METHOD  M_STATE_RESETTING
VAR_INPUT
END_VAR
Error :=_Error;
Done :=_Executed;
Busy := FALSE;


CASE uiResettingStep OF
	
	0:
		ConveyorMotor.M_MotorStop();
		M_RecoveryAllObjects();
		uiResettingStep:=9999;


	9999:
		M_RecoveryAllObjects();
		_ResetCompleted:=TRUE;
END_CASE
IF _ResetCompleted THEN
	eSTATE:=STATE_DORMANT;
END_IF
END_METHOD

END_FUNCTION_BLOCK

// ---- Library/20_MachineUnits/22_AllocateArea/Old_Version_Service/FB_OutRobot_EmptyBoxMove_old.TcPOU
FUNCTION_BLOCK FB_OutRobot_EmptyBoxMove_old EXTENDS FB_ObjectBase_V2
VAR_INPUT
//    Execute    :BOOL;   // True : This prog will start.
//    Abort      :BOOL;   // True : This prog will be abort.
//    Reset      :BOOL;   // True : This prog will be reset.
//    ObjectName :STRING; // Set this fb name(About it's action)
	INPUT            			   : REFERENCE TO ST_InputTable;
	Cylinder   					   : REFERENCE TO UNI_CylinderList;
	Motor      					   : REFERENCE TO UNI_MotorList;
	AutoMode_OutRobotMoveMove : st_AutoMode_ClampingBoxesJob;	
	Cylinders					   : REFERENCE TO ARRAY[0..1] OF FB_Cylinder;
	Clips						   : REFERENCE TO ARRAY[0..1] OF FB_Cylinder;
END_VAR

VAR_OUTPUT
//    Busy    :BOOL;        // True : This prog is running.
//    Done    :BOOL;        // True : Command has been executed.
//    Aborted :BOOL;        // True : This prog is aborted.
//    Error   :BOOL;        // True : This prog has an error.
//    ErrorID :UINT;       // Output ErrorID
//    Status  :T_MaxString; // Output this prog status by string(255bytes)
END_VAR

VAR
//    eState :E_MethodStatus_Basic;
//	uiExecutingStep : UDINT; // This var is used to been controll STATE_EXECUTING process.
//	uiResettingStep : UDINT;
//	uiAbortingStep : UDINT;
//	_Executed :BOOL; // Executing process completed.
//	_Error : BOOL; // FB has an error.
//	_ResetCompleted : BOOL; // FB resetting completed.
//	_AbortCompleted : BOOL; // FB aborting completed.
	//_Abort		: BOOL;
	strStatus	: STRING;
	uiResumeStep : UINT;
	tonTimeOut   :TON;
	tonTimeDelay   :TON;
	iWorkingIndex : INT;
	_UniqueErrorCode :STRING;	
	
	PickingPos	: ARRAY[0..1] OF ST_PositionTable;
	PlacingPos  : ARRAY[0..1] OF ST_PositionTable;
	PressCylinderOnI5			   : REFERENCE TO FB_Cylinder;
	bSyncPick	: BOOL;
	bSyncPlace	: BOOL;
	SensorOnConveyor		   : BIT;
	ConveyorMotor				   : REFERENCE TO FB_Motor;
	UseA	: BOOL;
	UseB	: BOOL;
END_VAR

A00_BasicUnits();
SUPER^.A10_StateControl();

ACTION A00_BasicUnits:
tonTimeOut(PT:=T#60S);
tonTimeDelay(PT:=T#1s);
END_ACTION

METHOD GetModelState
VAR_OUTPUT
    xDone    :BOOL;
    xBusy    :BOOL;
    xError   :BOOL;
    xAborted :BOOL;
    iErrorID :UDINT;
	UniqueErrorCode : STRING;
END_VAR
xDone    := Done;
xBusy    := Busy;
xError   := Error;
xAborted := Abort;
iErrorID := ErrorID;
UniqueErrorCode := THIS^.UniqueErrorCode;
END_METHOD

METHOD GetName : STRING
GetName := ObjectName;
END_METHOD

METHOD PRIVATE M_CheckCommand : BOOL
VAR_INPUT
END_VAR


M_CheckCommand := true;
END_METHOD

METHOD PRIVATE M_GetWorkingConditions : BOOL
VAR_INPUT
END_VAR
IF AutoMode_OutRobotMoveMove.ClampingInfo.UseClibA THEN
	PickingPos[0] :=FUN_GetPositionTableData('I',5,0);
	PlacingPos[0]:=FUN_GetPositionTableData('R',1,0);
	UseA :=TRUE;
END_IF

IF AutoMode_OutRobotMoveMove.ClampingInfo.UseClibB THEN
	PickingPos[1] :=FUN_GetPositionTableData('I',5,1);
	PlacingPos[1]:=FUN_GetPositionTableData('R',2,1);
	UseB := TRUE;
END_IF

IF PlacingPos[0].X_Pos =PlacingPos[1].X_Pos AND PlacingPos[0].Y_Pos = PlacingPos[1].Y_Pos AND UseA AND UseB  THEN
		bSyncPlace:=TRUE;
	ELSE
		bSyncPlace:=FALSE;	
END_IF
IF PickingPos[0].X_Pos =PickingPos[1].X_Pos AND PickingPos[0].Y_Pos = PickingPos[1].Y_Pos AND UseA AND UseB THEN
		bSyncPick:=TRUE;
	ELSE
		bSyncPick:=FALSE;	
END_IF

PressCylinderOnI5 REF= Cylinder.List.fbDifferentSizeCV_Press2;


ConveyorMotor REF= Motor.List.TransmitDifferentSideCV;
END_METHOD

METHOD PRIVATE M_RecoveryAllObjects : BOOL
VAR_INPUT
END_VAR
VAR 
	i : INT;
END_VAR
FOR i:=0 TO 1 DO
	IF Clips[i].xError THEN
		Clips[i].M_Reset();
		ELSE
		Clips[i].M_Retract();		
	END_IF
	IF Cylinders[i].xError THEN
	Cylinders[i].M_Reset();	
	ELSE
	Cylinders[i].M_Retract();	
	END_IF
END_FOR


IF arAxisCtrl_gb[AxisNo.OutRobot_X].Admin.Axis.Status.Error THEN

	arAxisCtrl_gb[AxisNo.OutRobot_X].Admin.ClearError:= TRUE;
ELSE
	arAxisCtrl_gb[AxisNo.OutRobot_X].Admin.ClearError:= FALSE;
END_IF

IF arAxisCtrl_gb[AxisNo.OutRobot_Y].Admin.Axis.Status.Error THEN

	arAxisCtrl_gb[AxisNo.OutRobot_Y].Admin.ClearError:= TRUE;
ELSE
	arAxisCtrl_gb[AxisNo.OutRobot_Y].Admin.ClearError:= FALSE;
END_IF
END_METHOD

METHOD  M_STATE_ABORTED
VAR_INPUT
END_VAR
ERROR :=TRUE;
Busy    := FALSE;
Aborted := TRUE;
Status := strStatus;

IF NOT Execute THEN
	eSTATE:=STATE_RESETTING;
END_IF

IF Execute AND Reset THEN
//	uiExecutingStep :=uiResumeStep;
	eSTATE:=STATE_EXECUTING;
END_IF
END_METHOD

METHOD  M_STATE_ABORTING
VAR_INPUT
END_VAR
VAR	 
 i : INT;
	bCylinderCheck: BOOL;
END_VAR
Error := TRUE;
CASE uiAbortingStep OF
	0 :
		bCylinderCheck :=TRUE;
		ConveyorMotor.M_MotorStop();
	
		FOR i :=0 TO 1 DO		
	    	Cylinders[i].M_Reset();
			Cylinders[i].M_Retract();
			bCylinderCheck:=bCylinderCheck AND Cylinders[i].InRearPosition;	
		END_FOR
		IF bCylinderCheck THEN		
			uiAbortingStep:=9999;
		END_IF
	9999:	_AbortCompleted:=TRUE;
END_CASE

IF _AbortCompleted THEN	
	eSTATE :=STATE_ABORTED;
END_IF
END_METHOD

METHOD  M_STATE_DONE
VAR_INPUT
END_VAR
Busy 	:= FALSE;
Done	:=TRUE;

IF NOT Execute THEN
	eSTATE:=STATE_RESETTING;
END_IF
END_METHOD

METHOD  M_STATE_DORMANT
VAR_INPUT
END_VAR
Busy            := FALSE;
Done            := FALSE;
Aborted         := FALSE;
Error           := FALSE;
ErrorID         := 0;
Status          := '';
_ResetCompleted := FALSE;
_Error          := FALSE;
_Executed       := FALSE;
_Abort	 :=FALSE;
strStatus :='FB_OutRobot_EmptyBoxMove: No Error';
uiExecutingStep :=uiResettingStep :=uiResumeStep :=0;
tonTimeOut.IN :=TRUE;
_UniqueErrorCode:='0';
iWorkingIndex :=0;
bSyncPlace := FALSE;
UseA := FALSE;
UseB :=FALSE;
IF Execute THEN
	eSTATE:=STATE_EXECUTING;
END_IF
END_METHOD

METHOD  M_STATE_ERROR
VAR_INPUT
END_VAR
ERROR   :=TRUE;
Busy	:=FALSE;
Status := strStatus;
IF __ISVALIDREF(ConveyorMotor) THEN
	ConveyorMotor.M_MotorStop();
END_IF
IF NOT Execute THEN	
eSTATE:=STATE_RESETTING;
END_IF
END_METHOD

METHOD  M_STATE_EXECUTING
VAR_INPUT
END_VAR
VAR_INST
	bMoveConveyorForward : BOOL;
	bMoveConveyorBackrward : BOOL;

END_VAR

VAR
	bCylinderCheck : BOOL := TRUE;
END_VAR
Busy :=TRUE;
SensorOnConveyor := INPUT.bDifferentSizeCV_BoxDetect5_Sensor;
IF bMoveConveyorForward THEN
	IF NOT ConveyorMotor.InBackWard THEN
		ConveyorMotor.M_MoveForward();
	END_IF
END_IF
IF bMoveConveyorBackrward THEN
	IF NOT ConveyorMotor.InForWard THEN
		ConveyorMotor.M_MoveBackward();
	END_IF
END_IF
CASE uiExecutingStep OF
	

0: //Idle
	bMoveConveyorForward:=FALSE;
	bMoveConveyorBackrward:=FALSE;
	tonTimeDelay.IN :=FALSE;
	tonTimeOut.IN := FALSE;
	iWorkingIndex :=0;
	M_GetWorkingConditions();
	
	
	M_RecoveryAllObjects();
	uiExecutingStep := 100;
	
100: //Check command
	
	IF PressCylinderOnI5.xError THEN
		PressCylinderOnI5.M_Reset();
	ELSE
		PressCylinderOnI5.M_Retract();
	END_IF
	
	IF M_CheckCommand() THEN
		uiExecutingStep:=200;
	END_IF
	
200: // Check No boxes turntable

	IF (UseA AND INPUT.bTurnTable_R1Detect_Sensor) OR (UseB AND INPUT.bTurnTable_R2Detect_Sensor) THEN
		_Abort:=TRUE;
		strStatus :='FB_OutRobot_EmptyBoxMove Step 200: Box On Turntable';
	ELSE
		IF UseA THEN
			iWorkingIndex :=0;
		ELSE
			iWorkingIndex :=1;	
		END_IF
		
		uiExecutingStep:=1000;	
	END_IF

	
1000: 
	// Move Conveyor
	// Move OutRobot to First clip picking	
	 //ConveyorMotor.M_MoveForward();
	 bMoveConveyorForward:=TRUE;
	arAxisCtrl_gb[AxisNo.OutRobot_X].PosMode.Position := PickingPos[iWorkingIndex].X_Pos;		
	arAxisCtrl_gb[AxisNo.OutRobot_Y].PosMode.Position := PickingPos[iWorkingIndex].Y_Pos;	
		IF ConveyorMotor.InForWard THEN
			uiExecutingStep:=1100;
		END_IF
		
1100://CheckSensor
	tonTimeDelay.IN:=SensorOnConveyor;
	
			
	IF tonTimeDelay.Q THEN
		tonTimeOut.IN :=FALSE;
		uiExecutingStep:=1200;
		tonTimeDelay.IN := FALSE;
		
	END_IF
	
	tonTimeOut.IN := TRUE;
	IF tonTimeOut.Q THEN
		tonTimeOut.IN :=FALSE;
		_Abort := TRUE;
		strStatus :='FB_OutRobot_EmptyBoxMove Step 1100: No Box on conveyor';
	END_IF

1200: //Press seconde box
	  PressCylinderOnI5.M_Extend();
	  IF PressCylinderOnI5.InFrontPosition THEN
		  tonTimeOut.IN :=FALSE;
		  uiExecutingStep:=1300;
	  END_IF
	  
	  	tonTimeOut.IN := TRUE;
	IF tonTimeOut.Q THEN
		tonTimeOut.IN :=FALSE;
		_Abort := TRUE;
		strStatus :='FB_OutRobot_EmptyBoxMove Step 1200: Block box on conveyor timeout';
	END_IF
	
1300: // Stop conveyor
	ConveyorMotor.M_MotorStop();
	bMoveConveyorForward:=FALSE;
	bMoveConveyorBackrward:=FALSE;
	IF ConveyorMotor.InStopped THEN
		 uiExecutingStep:=1400;
	END_IF

1400: // Check outRobot arrived
	IF		(arAxisStatus_gb[AxisNo.OutRobot_X].Admin._OpModeAck = ModePosAbs AND arAxisStatus_gb[AxisNo.OutRobot_X].Admin.CmdDone) 
	AND (arAxisStatus_gb[AxisNo.OutRobot_Y].Admin._OpModeAck = ModePosAbs AND arAxisStatus_gb[AxisNo.OutRobot_Y].Admin.CmdDone) 
	THEN
		tonTimeOut.IN :=FALSE;
		uiExecutingStep:=1500;
	END_IF	
	
	tonTimeOut.IN := TRUE;
	IF tonTimeOut.Q THEN
		tonTimeOut.IN :=FALSE;
		_Error := TRUE;
		strStatus :='FB_OutRobot_EmptyBoxMove Step 1400: Move robot to picking position timeout';
	END_IF
	
1500: //Clip Down Pick
	 Cylinders[iWorkingIndex].M_Extend();
	  IF Cylinders[iWorkingIndex].InFrontPosition THEN
		  tonTimeOut.IN :=FALSE;
		  uiExecutingStep:=1700;
	  END_IF
	
	 tonTimeOut.IN := TRUE;
	IF tonTimeOut.Q THEN
		tonTimeOut.IN :=FALSE;
		_Abort := TRUE;
		strStatus :='FB_OutRobot_EmptyBoxMove Step 1500: Cylinder pick down timeout';
	END_IF
	
1700: // Clip close Pick
	Clips[iWorkingIndex].M_Extend();
	  IF Clips[iWorkingIndex].InFrontPosition THEN
		  tonTimeOut.IN :=FALSE;
		  uiExecutingStep:=1800;
	  END_IF
	  
	   tonTimeOut.IN := TRUE;
	IF tonTimeOut.Q THEN
		tonTimeOut.IN :=FALSE;
		_Abort := TRUE;
		strStatus :='FB_OutRobot_EmptyBoxMove Step 1700: clip pick close timeout';
	END_IF

1800: // Clip Up Pick
	   Cylinders[iWorkingIndex].M_Retract();
	  IF Cylinders[iWorkingIndex].InRearPosition THEN
		  
		  tonTimeOut.IN :=FALSE;
		  uiExecutingStep:=1850;
	  END_IF
	  
	    tonTimeOut.IN := TRUE;
	IF tonTimeOut.Q THEN
		tonTimeOut.IN :=FALSE;
		_Abort := TRUE;
		strStatus :='FB_OutRobot_EmptyBoxMove Step 1800: cylinder pick up timeout';
	END_IF
1850: //Check box leave
		IF NOT SensorOnConveyor THEN
			PressCylinderOnI5.M_Retract();
			uiExecutingStep:=1900;
		else
			_Error := TRUE;
			strStatus :='FB_OutRobot_EmptyBoxMove Step 1850: Box still on conveyor';
		END_IF
		
1900: // If Next pick
	  IF iWorkingIndex>=1 OR NOT UseB THEN
		  IF UseA THEN
		  	iWorkingIndex :=0;
		  ELSIF UseB THEN
			iWorkingIndex :=1;	
		  END_IF
		  uiExecutingStep:=2000;
		  //Go to placing box
	  ELSIF  iWorkingIndex=0 AND UseB THEN
			iWorkingIndex:=iWorkingIndex+1;
	 		uiExecutingStep:=1000;
	  END_IF
	  
2000: // Move to Placing pos
	 arAxisCtrl_gb[AxisNo.OutRobot_X].PosMode.Position := PlacingPos[iWorkingIndex].X_Pos;		
	 arAxisCtrl_gb[AxisNo.OutRobot_Y].PosMode.Position := PlacingPos[iWorkingIndex].Y_Pos;	
	 uiExecutingStep:=2100;

2100: // Waiting outRobot move to placing pos	 
	 IF	(arAxisStatus_gb[AxisNo.OutRobot_X].Admin._OpModeAck = ModePosAbs AND arAxisStatus_gb[AxisNo.OutRobot_X].Admin.CmdDone) 
	AND (arAxisStatus_gb[AxisNo.OutRobot_Y].Admin._OpModeAck = ModePosAbs AND arAxisStatus_gb[AxisNo.OutRobot_Y].Admin.CmdDone) 
	THEN
		tonTimeOut.IN :=FALSE;
		uiExecutingStep:=2200;
	END_IF	

	    tonTimeOut.IN := TRUE;
	IF tonTimeOut.Q THEN
		tonTimeOut.IN :=FALSE;
		_Error := TRUE;
		strStatus :='FB_OutRobot_EmptyBoxMove Step 2100: Move robot to placing position timeout';
	END_IF
	
2200: //Cllp Down place
	bCylinderCheck := TRUE;
	Cylinders[iWorkingIndex].M_Extend();
	bCylinderCheck :=Cylinders[iWorkingIndex].InFrontPosition AND bCylinderCheck;
	IF bSyncPlace THEN
		Cylinders[1].M_Extend();
		bCylinderCheck :=Cylinders[1].InFrontPosition AND bCylinderCheck;
	END_IF	
	 
	IF bCylinderCheck THEN
		tonTimeOut.IN :=FALSE;
		uiExecutingStep:=2300;
	END_IF 
	
	   tonTimeOut.IN := TRUE;
	IF tonTimeOut.Q THEN
		tonTimeOut.IN :=FALSE;
		_Abort := TRUE;
		strStatus :='FB_OutRobot_EmptyBoxMove Step 2200: Cylinder place down timeout';
	END_IF
	
2300: // Clip open Place
	bCylinderCheck := TRUE;
	Clips[iWorkingIndex].M_Retract();
	bCylinderCheck := Clips[iWorkingIndex].InRearPosition AND bCylinderCheck;
	IF bSyncPlace THEN
		Clips[1].M_Retract();
		bCylinderCheck := Clips[1].InRearPosition AND bCylinderCheck;
	END_IF	
	 
	IF bCylinderCheck THEN
		tonTimeOut.IN :=FALSE;
		uiExecutingStep:=2400;
	END_IF 
	  
	  tonTimeOut.IN := TRUE;
	IF tonTimeOut.Q THEN
		tonTimeOut.IN :=FALSE;
		_Abort := TRUE;
		strStatus :='FB_OutRobot_EmptyBoxMove Step 2300: clip place open timeout';
	END_IF
	  
2400: // Clip up Placing
	bCylinderCheck := TRUE;
	Cylinders[iWorkingIndex].M_Retract();
	bCylinderCheck :=Cylinders[iWorkingIndex].InRearPosition AND bCylinderCheck;
	IF bSyncPlace THEN
		Cylinders[1].M_Retract();
		bCylinderCheck :=Cylinders[1].InRearPosition AND bCylinderCheck;
	END_IF	
	 
	IF bCylinderCheck THEN
		tonTimeOut.IN :=FALSE;
		uiExecutingStep:=2500;
	END_IF 
	  tonTimeOut.IN := TRUE;
	IF tonTimeOut.Q THEN
		tonTimeOut.IN :=FALSE;
		_Abort := TRUE;
		strStatus :='FB_OutRobot_EmptyBoxMove Step 2400: cylinder place up timeout';
	END_IF
	
2500: // If Next place
	IF iWorkingIndex>=1 OR bSyncPlace OR NOT UseB THEN
		uiExecutingStep:=2600;
		// Finish
	ELSE	
		iWorkingIndex := iWorkingIndex+1;
	  	uiExecutingStep:=2000;
	END_IF
2600: //Check box on turntable

	IF (UseA AND NOT INPUT.bTurnTable_R1Detect_Sensor) OR (UseB AND NOT INPUT.bTurnTable_R2Detect_Sensor) THEN
		_Error:=TRUE;
		strStatus :='FB_OutRobot_EmptyBoxMove Step 2600: Box not On Turntable';
	ELSE
		uiExecutingStep:=3000;
	END_IF
3000: // Finish	
	bMoveConveyorForward:=FALSE;
	bMoveConveyorBackrward:=FALSE;
	_Executed:=TRUE;
	
END_CASE
	
IF NOT Execute THEN
	eState:=STATE_RESETTING;
END_IF
IF _Error THEN
	eState:=STATE_ERROR;
END_IF
IF _Abort THEN
	eSTATE:=STATE_ABORTING;
END_IF
IF _Executed THEN
	eSTATE:=STATE_Done;
END_IF
END_METHOD

METHOD  M_STATE_RESETTING
VAR_INPUT
END_VAR
Error :=_Error;
Done :=_Executed;
Busy := FALSE;


CASE uiResettingStep OF
	
	0:
		uiResettingStep:=9999;
		ConveyorMotor.M_MotorStop();
		M_RecoveryAllObjects();
		IF PressCylinderOnI5.xError THEN
		PressCylinderOnI5.M_Reset();
	ELSE
		PressCylinderOnI5.M_Retract();
	END_IF

	9999:
		_ResetCompleted:=TRUE;
END_CASE
IF _ResetCompleted THEN
	eSTATE:=STATE_DORMANT;
END_IF
END_METHOD

END_FUNCTION_BLOCK

// ---- Library/20_MachineUnits/22_AllocateArea/Old_Version_Service/FB_OutRobot_RareBoxMove_old.TcPOU
FUNCTION_BLOCK FB_OutRobot_RareBoxMove_old EXTENDS FB_ObjectBase_V2
VAR_INPUT
//    Execute    :BOOL;   // True : This prog will start.
//    Abort      :BOOL;   // True : This prog will be abort.
//    Reset      :BOOL;   // True : This prog will be reset.
//    ObjectName :STRING; // Set this fb name(About it's action)
	INPUT            			   : REFERENCE TO ST_InputTable;	
	Cylinder   					   : REFERENCE TO UNI_CylinderList;
	Motor      					   : REFERENCE TO UNI_MotorList;
	Cylinders					   : REFERENCE TO ARRAY[0..1] OF FB_Cylinder;
	Clips						   : REFERENCE TO ARRAY[0..1] OF FB_Cylinder;
	AutoMode_OutRobotMoveMove : st_AutoMode_ClampingBoxesJob;	
END_VAR

VAR_OUTPUT
//    Busy    :BOOL;        // True : This prog is running.
//    Done    :BOOL;        // True : Command has been executed.
//    Aborted :BOOL;        // True : This prog is aborted.
//    Error   :BOOL;        // True : This prog has an error.
//    ErrorID :UINT;       // Output ErrorID
//    Status  :T_MaxString; // Output this prog status by string(255bytes)
END_VAR

VAR
//    eState :E_MethodStatus_Basic;
//	uiExecutingStep : UDINT; // This var is used to been controll STATE_EXECUTING process.
//	uiResettingStep : UDINT;
//	uiAbortingStep : UDINT;
//	_Executed :BOOL; // Executing process completed.
//	_Error : BOOL; // FB has an error.
//	_ResetCompleted : BOOL; // FB resetting completed.
//	_AbortCompleted : BOOL; // FB aborting completed.
	//_Abort		: BOOL;
	strStatus	: STRING;
	uiResumeStep : UINT;
	tonTimeOut   :TON;
	tonTimeDelay   :TON;
	iWorkingIndex : INT;
	_UniqueErrorCode :STRING;	
	PickingPos	: ARRAY[0..1] OF ST_PositionTable;
	PlacingPos  : ARRAY[0..1] OF ST_PositionTable;
	bSyncPick	: BOOL;
	bSyncPlace	: BOOL;
	SensorOnConveyor			   : BIT;
	ConveyorMotor				   : REFERENCE TO FB_Motor;
	UseA	: BOOL;
	UseB	: BOOL;
	bMotorMoveForward : BOOL;	
		
	// check position
	bSamePosX	: BOOL;
	bSamePosY	: BOOL;
	lrEpsPos 	: LREAL := 0.001;
END_VAR

A00_BasicUnits();
SUPER^.A10_StateControl();

ACTION A00_BasicUnits:
tonTimeOut(PT:=T#60S);
tonTimeDelay(PT:=T#1.5s);
END_ACTION

METHOD GetModelState
VAR_OUTPUT
    xDone    :BOOL;
    xBusy    :BOOL;
    xError   :BOOL;
    xAborted :BOOL;
    iErrorID :UDINT;
	UniqueErrorCode : STRING;
END_VAR
xDone    := Done;
xBusy    := Busy;
xError   := Error;
xAborted := Abort;
iErrorID := ErrorID;
UniqueErrorCode := THIS^.UniqueErrorCode;
END_METHOD

METHOD GetName : STRING
GetName := ObjectName;
END_METHOD

METHOD PRIVATE M_CheckCommand : BOOL
VAR_INPUT
END_VAR


M_CheckCommand := true;
END_METHOD

METHOD PRIVATE M_GetWorkingConditions : BOOL
VAR_INPUT
END_VAR
//For rare box move , Boxes must place on same position , therefor only work with TargetPosition of ClipA

IF AutoMode_OutRobotMoveMove.ClampingInfo.TargetOfClipA = 5 THEN	
	ConveyorMotor REF= Motor.List.TransmitDifferentSideCV;
ELSIF AutoMode_OutRobotMoveMove.ClampingInfo.TargetOfClipA = 6 THEN
	ConveyorMotor REF= Motor.List.TransmitSameSideCV;
ELSIF AutoMode_OutRobotMoveMove.ClampingInfo.TargetOfClipA = 3 THEN
	ConveyorMotor REF= Motor.List.TransmitDifferentSideCV;
ELSIF AutoMode_OutRobotMoveMove.ClampingInfo.TargetOfClipA = 4 THEN
	ConveyorMotor REF= Motor.List.TransmitSameSideCV;	
END_IF

IF AutoMode_OutRobotMoveMove.ClampingInfo.TargetOfClipA=5 OR AutoMode_OutRobotMoveMove.ClampingInfo.TargetOfClipA=6 THEN
		bMotorMoveForward := FALSE;
	ELSE
		bMotorMoveForward := TRUE;	
END_IF
IF AutoMode_OutRobotMoveMove.ClampingInfo.UseClibA THEN
	PickingPos[0] :=FUN_GetPositionTableData('R',1,0);
	UseA := TRUE;
	CASE  AutoMode_OutRobotMoveMove.ClampingInfo.TargetOfClipA OF	
		
	3,4:
		PlacingPos[0] :=FUN_GetPositionTableData('O',AutoMode_OutRobotMoveMove.ClampingInfo.TargetOfClipA,0);
	5,6:
		PlacingPos[0] :=FUN_GetPositionTableData('I',AutoMode_OutRobotMoveMove.ClampingInfo.TargetOfClipA,0);
	ELSE
		strStatus :='FB_OutRobot_RareBoxMove: Wrong command: Clip A target not allow';
		M_GetWorkingConditions := FALSE;
		RETURN;
	END_CASE
END_IF

IF AutoMode_OutRobotMoveMove.ClampingInfo.UseClibB THEN
	PickingPos[1] :=FUN_GetPositionTableData('R',2,1);
	UseB :=TRUE;
	CASE AutoMode_OutRobotMoveMove.ClampingInfo.TargetOfClipA OF
		
	3,4:
		PlacingPos[1] :=FUN_GetPositionTableData('O',AutoMode_OutRobotMoveMove.ClampingInfo.TargetOfClipA,1);
	5,6 :
		PlacingPos[1] :=FUN_GetPositionTableData('I',AutoMode_OutRobotMoveMove.ClampingInfo.TargetOfClipA,1);
	ELSE
		strStatus :='FB_OutRobot_RareBoxMove: Wrong command: Clip B target not allow';
		M_GetWorkingConditions := FALSE;
		RETURN;
	END_CASE
END_IF

IF PlacingPos[0].X_Pos =PlacingPos[1].X_Pos AND PlacingPos[0].Y_Pos = PlacingPos[1].Y_Pos AND UseA AND UseB THEN
		bSyncPlace:=TRUE;
	ELSE
		bSyncPlace:=FALSE;	
END_IF

bSamePosX := ABS(PickingPos[0].X_Pos - PickingPos[1].X_Pos) < lrEpsPos;
bSamePosY := ABS(PickingPos[0].Y_Pos - PickingPos[1].Y_Pos) < lrEpsPos;
IF bSamePosX AND bSamePosY AND UseA AND UseB THEN
		bSyncPick:=TRUE;
	ELSE
		bSyncPick:=FALSE;	
END_IF

M_GetWorkingConditions :=TRUE;
END_METHOD

METHOD PRIVATE M_RecoveryAllObjects : BOOL
VAR_INPUT
END_VAR
VAR 
	i : INT;
END_VAR
FOR i:=0 TO 1 DO
	IF Clips[i].xError THEN
		Clips[i].M_Reset();
		ELSE
		Clips[i].M_Retract();		
	END_IF
	IF Cylinders[i].xError THEN
	Cylinders[i].M_Reset();	
	ELSE
	Cylinders[i].M_Retract();	
	END_IF
END_FOR

IF arAxisCtrl_gb[AxisNo.OutRobot_X].Admin.Axis.Status.Error THEN

	arAxisCtrl_gb[AxisNo.OutRobot_X].Admin.ClearError:= TRUE;
ELSE
	arAxisCtrl_gb[AxisNo.OutRobot_X].Admin.ClearError:= FALSE;
END_IF

IF arAxisCtrl_gb[AxisNo.OutRobot_Y].Admin.Axis.Status.Error THEN

	arAxisCtrl_gb[AxisNo.OutRobot_Y].Admin.ClearError:= TRUE;
ELSE
	arAxisCtrl_gb[AxisNo.OutRobot_Y].Admin.ClearError:= FALSE;
END_IF
END_METHOD

METHOD PRIVATE M_SensorUpdate : BOOL
VAR_INPUT
END_VAR
IF AutoMode_OutRobotMoveMove.ClampingInfo.TargetOfClipA = 5 THEN
	SensorOnConveyor := INPUT.bDifferentSizeCV_BoxDetect5_Sensor;
ELSIF AutoMode_OutRobotMoveMove.ClampingInfo.TargetOfClipA = 6 THEN
	SensorOnConveyor := INPUT.bSameSizeCV_BoxDetect5_Sensor;
ELSIF AutoMode_OutRobotMoveMove.ClampingInfo.TargetOfClipA = 3 THEN
	SensorOnConveyor := INPUT.bDifferentSizeCV_BoxDetect4_Sensor;
ELSIF AutoMode_OutRobotMoveMove.ClampingInfo.TargetOfClipA = 4 THEN
	SensorOnConveyor := INPUT.bSameSizeCV_BoxDetect4_Sensor;	
END_IF
END_METHOD

METHOD  M_STATE_ABORTED
VAR_INPUT
END_VAR
ERROR :=TRUE;
Busy    := FALSE;
Aborted := TRUE;
Status := strStatus;

IF NOT Execute THEN
	eSTATE:=STATE_RESETTING;
END_IF

IF Execute AND Reset THEN
//	uiExecutingStep :=uiResumeStep;
	eSTATE:=STATE_EXECUTING;
END_IF
END_METHOD

METHOD  M_STATE_ABORTING
VAR_INPUT
END_VAR
VAR	
	i : INT;
	bCylinderCheck : BOOL :=true;
END_VAR
CASE uiAbortingStep OF
	0 :
		ConveyorMotor.M_MotorStop();
		bCylinderCheck := TRUE;
		FOR i :=0 TO 1 DO		
	    	Cylinders[i].M_Reset();
			Cylinders[i].M_Retract();
			bCylinderCheck:=bCylinderCheck AND Cylinders[i].InRearPosition;	
		END_FOR
		IF bCylinderCheck THEN		
			uiAbortingStep:=9999;
		END_IF
	9999:	
	_Abort := FALSE;
		_AbortCompleted:=TRUE;
END_CASE

IF _AbortCompleted THEN	
	eSTATE :=STATE_ABORTED;
END_IF
END_METHOD

METHOD  M_STATE_DONE
VAR_INPUT
END_VAR
Busy 	:= FALSE;
Done	:=TRUE;

IF NOT Execute THEN
	eSTATE:=STATE_RESETTING;
END_IF
END_METHOD

METHOD  M_STATE_DORMANT
VAR_INPUT
END_VAR
Busy            := FALSE;
Done            := FALSE;
Aborted         := FALSE;
Error           := FALSE;
ErrorID         := 0;
Status          := '';
_ResetCompleted := FALSE;
_Error          := FALSE;
_Executed       := FALSE;
strStatus :='FB_OutRobot_RareBoxMove: No Error';
uiExecutingStep :=uiResettingStep :=uiResumeStep :=0;
tonTimeOut.IN :=TRUE;
_UniqueErrorCode:='0';
iWorkingIndex :=0;
bSyncPick :=FALSE;
bSyncPlace := FALSE;
UseA := FALSE;
UseB :=FALSE;
bMotorMoveForward := FALSE;
_Abort :=FALSE;
_Error := FALSE;
bSamePosX := FALSE;
bSamePosY := FALSE;

IF Execute THEN
	eSTATE:=STATE_EXECUTING;
END_IF
END_METHOD

METHOD  M_STATE_ERROR
VAR_INPUT
END_VAR
ERROR   :=TRUE;
Busy	:=FALSE;
Status := strStatus;
IF __ISVALIDREF(ConveyorMotor) THEN
	ConveyorMotor.M_MotorStop();
END_IF
IF NOT Execute THEN	
eSTATE:=STATE_RESETTING;
END_IF
END_METHOD

METHOD  M_STATE_EXECUTING
VAR_INPUT
END_VAR
VAR_INST
	bMoveConveyorForward : BOOL;
	bMoveConveyorBackrward : BOOL;

END_VAR

VAR
	bCylinderCheck : BOOL := TRUE;
END_VAR
Busy :=TRUE;
M_SensorUpdate();
IF bMoveConveyorForward THEN
	IF NOT ConveyorMotor.InBackWard THEN
		ConveyorMotor.M_MoveForward();	
	END_IF	
END_IF

IF bMoveConveyorBackrward THEN
	IF NOT ConveyorMotor.InForWard THEN
		ConveyorMotor.M_MoveBackward();
	END_IF
END_IF
CASE uiExecutingStep OF
	

0: //Idle
	bMoveConveyorForward:=FALSE;
	tonTimeDelay.IN :=FALSE;
	tonTimeOut.IN := FALSE;
	iWorkingIndex :=0;	
	
	M_RecoveryAllObjects();
	uiExecutingStep := 100;
	
100: //Check command
	IF M_GetWorkingConditions()THEN	
		uiExecutingStep:=200;
	ELSE
		_Error :=TRUE;
	END_IF
	
200: // Check  boxes on turntable

	IF (UseA AND NOT INPUT.bTurnTable_R1Detect_Sensor) OR (UseB AND NOT INPUT.bTurnTable_R2Detect_Sensor) THEN
		_Error:=TRUE;
		strStatus :='FB_OutRobot_RareBoxMove Step 200: Box Not on Turntable';
	ELSE
		IF UseA THEN
			iWorkingIndex :=0;
		ELSE
			iWorkingIndex :=1;	
		END_IF
		
		uiExecutingStep:=1000;	
	END_IF

	
1000: 
	// Move OutRobot to First clip picking	
	 	 
	arAxisCtrl_gb[AxisNo.OutRobot_X].PosMode.Position := PickingPos[iWorkingIndex].X_Pos;		
	arAxisCtrl_gb[AxisNo.OutRobot_Y].PosMode.Position := PickingPos[iWorkingIndex].Y_Pos;	
	uiExecutingStep:=1100;
		// todo : Check axes is moving
1100:
	// Check outRobot arrived
	IF		(arAxisStatus_gb[AxisNo.OutRobot_X].Admin._OpModeAck = ModePosAbs AND arAxisStatus_gb[AxisNo.OutRobot_X].Admin.CmdDone) 
	AND (arAxisStatus_gb[AxisNo.OutRobot_Y].Admin._OpModeAck = ModePosAbs AND arAxisStatus_gb[AxisNo.OutRobot_Y].Admin.CmdDone) 
	THEN
		tonTimeOut.IN := FALSE;
		uiExecutingStep:=1200;
	END_IF	
	tonTimeOut.IN := TRUE;
	IF tonTimeOut.Q THEN
		tonTimeOut.IN := FALSE;
		_Error :=TRUE;
		strStatus :='FB_OutRobot_RareBoxMove Step 1100: Robot move to picking position timeout';
	END_IF
	
1200: //Clip Down Pick	  
	bCylinderCheck := TRUE;
	Cylinders[iWorkingIndex].M_Extend();
	bCylinderCheck := Cylinders[iWorkingIndex].InFrontPosition AND bCylinderCheck;
	IF bSyncPick THEN
		Cylinders[1].M_Extend();
		bCylinderCheck := Cylinders[1].InFrontPosition AND bCylinderCheck;
	END_IF	
	 
	IF bCylinderCheck THEN
		tonTimeOut.IN := FALSE;
		uiExecutingStep:=1300;
	END_IF 
	tonTimeOut.IN := TRUE;
	IF tonTimeOut.Q THEN
		tonTimeOut.IN := FALSE;
		_Abort :=TRUE;
		strStatus :='FB_OutRobot_RareBoxMove Step 1200: Cylinder pick down timeout';
	END_IF
	
1300: // Clip close Pick
	bCylinderCheck := TRUE;
	Clips[iWorkingIndex].M_Extend();
	bCylinderCheck := Clips[iWorkingIndex].InFrontPosition AND bCylinderCheck;
	IF bSyncPick THEN
		Clips[1].M_Extend();
		bCylinderCheck := Clips[1].InFrontPosition AND bCylinderCheck;
	END_IF	
	 
	IF bCylinderCheck THEN
		tonTimeOut.IN := FALSE;
		uiExecutingStep:=1400;
	END_IF 
	
		tonTimeOut.IN := TRUE;
	IF tonTimeOut.Q THEN
		tonTimeOut.IN := FALSE;
		_Abort :=TRUE;
		strStatus :='FB_OutRobot_RareBoxMove Step 1300: clip pick close timeout';
	END_IF
	
1400: // Clip Up Pick
	bCylinderCheck := TRUE;
	Cylinders[iWorkingIndex].M_Retract();
	bCylinderCheck := Cylinders[iWorkingIndex].InRearPosition AND bCylinderCheck;
	IF bSyncPick THEN
		Cylinders[1].M_Retract();
		bCylinderCheck := Cylinders[1].InRearPosition AND bCylinderCheck;
	END_IF	
	 
	IF bCylinderCheck THEN
		tonTimeOut.IN := FALSE;
		uiExecutingStep:=1500;
	END_IF 
	
		tonTimeOut.IN := TRUE;
	IF tonTimeOut.Q THEN
		tonTimeOut.IN := FALSE;
		_Abort :=TRUE;
		strStatus :='FB_OutRobot_RareBoxMove Step 1400: cylinder pick up timeout';
	END_IF
	  
1500: // If Next pick
	  IF iWorkingIndex>=1 OR bSyncPick OR NOT UseB THEN
		//Go to placing step
			IF UseA THEN
				iWorkingIndex:=0;
			ELSE
				iWorkingIndex:=1;	
			END_IF
			uiExecutingStep:=1600;
		ELSE
			iWorkingIndex :=iWorkingIndex +1;
			uiExecutingStep:=1000;	
	  END_IF
	  
1600: // Check box
		
	IF (UseA AND  INPUT.bTurnTable_R1Detect_Sensor) OR (UseB AND  INPUT.bTurnTable_R2Detect_Sensor) THEN
		
		//
	ELSE
		tonTimeOut.IN := FALSE;
		uiExecutingStep:=2000;
	END_IF
		tonTimeOut.IN := TRUE;
	IF tonTimeOut.Q THEN
		tonTimeOut.IN := FALSE;
		_Error :=TRUE;
		strStatus :='FB_OutRobot_RareBoxMove Step 1600: Box still on Turntable';
	END_IF

2000: // Move to Placing pos
	  // Move Conveyor 
	  IF bMotorMoveForward THEN
		bMoveConveyorForward:=TRUE;
	  ELSE	 
		 bMoveConveyorBackrward:=TRUE; 
	 	 ConveyorMotor.M_MoveBackward(); 
	  END_IF
	 
	 arAxisCtrl_gb[AxisNo.OutRobot_X].PosMode.Position := PlacingPos[iWorkingIndex].X_Pos;		
	 arAxisCtrl_gb[AxisNo.OutRobot_Y].PosMode.Position := PlacingPos[iWorkingIndex].Y_Pos;	
	 uiExecutingStep:=2100;

2100: // Waiting outRobot move to placing pos	 
	  // Check sensor off for a while
	tonTimeDelay.IN := NOT 	SensorOnConveyor;
	 IF	(arAxisStatus_gb[AxisNo.OutRobot_X].Admin._OpModeAck = ModePosAbs AND arAxisStatus_gb[AxisNo.OutRobot_X].Admin.CmdDone) 
	AND (arAxisStatus_gb[AxisNo.OutRobot_Y].Admin._OpModeAck = ModePosAbs AND arAxisStatus_gb[AxisNo.OutRobot_Y].Admin.CmdDone)
	AND  tonTimeDelay.Q
	THEN		
		tonTimeOut.IN := FALSE;
		uiExecutingStep:=2150;
	END_IF	

		tonTimeOut.IN := TRUE;
	IF tonTimeOut.Q THEN
		tonTimeOut.IN := FALSE;
		_Error :=TRUE;
		strStatus :='FB_OutRobot_RareBoxMove Step 2100: robot move to placing position timeout';
	END_IF
	
2150 : //Motor stop
		tonTimeDelay.IN := FALSE;
		bMoveConveyorForward := FALSE;
		bMoveConveyorBackrward:=FALSE;
		ConveyorMotor.M_MotorStop();
		uiExecutingStep:=2200;
		

2200: //Cllp Down place
	bCylinderCheck := TRUE;
	Cylinders[iWorkingIndex].M_Extend();
	bCylinderCheck := Cylinders[iWorkingIndex].InFrontPosition AND bCylinderCheck;
	IF bSyncPlace THEN
		Cylinders[1].M_Extend();
		bCylinderCheck := Cylinders[1].InFrontPosition AND bCylinderCheck;
	END_IF	
	 
	IF bCylinderCheck THEN
		tonTimeOut.IN := FALSE;
		uiExecutingStep:=2300;
	END_IF 
		tonTimeOut.IN := TRUE;
	IF tonTimeOut.Q THEN
		tonTimeOut.IN := FALSE;
		_Abort :=TRUE;
		strStatus :='FB_OutRobot_RareBoxMove Step 2200: Cylinder place down timeout';
	END_IF
	
2300: // Clip open Place
	bCylinderCheck := TRUE;
	Clips[iWorkingIndex].M_Retract();
	bCylinderCheck := Clips[iWorkingIndex].InRearPosition AND bCylinderCheck;
	IF bSyncPlace THEN
		Clips[1].M_Retract();
		bCylinderCheck := Clips[1].InRearPosition AND bCylinderCheck;
	END_IF	
	 
	IF bCylinderCheck THEN
		tonTimeOut.IN := FALSE;
		uiExecutingStep:=2400;
	END_IF 
	  
		tonTimeOut.IN := TRUE;
	IF tonTimeOut.Q THEN
		tonTimeOut.IN := FALSE;
		_Abort :=TRUE;
		strStatus :='FB_OutRobot_RareBoxMove Step 2300: clip place open timeout';
	END_IF
	  
2400: // Clip up Placing
	bCylinderCheck := TRUE;
	Cylinders[iWorkingIndex].M_Retract();
	bCylinderCheck := Cylinders[iWorkingIndex].InRearPosition AND bCylinderCheck;
	IF bSyncPlace THEN
		Cylinders[1].M_Retract();
		bCylinderCheck := Cylinders[1].InRearPosition AND bCylinderCheck;
	END_IF	
	 
	IF bCylinderCheck THEN
		tonTimeOut.IN := FALSE;
		uiExecutingStep:=2500;
	END_IF 
		tonTimeOut.IN := TRUE;
	IF tonTimeOut.Q THEN
		tonTimeOut.IN := FALSE;
		_Abort :=TRUE;
		strStatus :='FB_OutRobot_RareBoxMove Step 2400: cylinder place up timeout';
	END_IF
	
2500: // If Next place
	IF iWorkingIndex>=1 OR bSyncPlace OR NOT UseB THEN
		uiExecutingStep:=2600;
		// Finish
	ELSE	
		iWorkingIndex := iWorkingIndex+1;
	  	uiExecutingStep:=2000;
	END_IF
	
2600: // Move conveyor a bit
		 IF bMotorMoveForward THEN
			 bMoveConveyorForward:=TRUE;		 
			 ConveyorMotor.M_MoveForward();
		  ELSE	 
			  bMoveConveyorBackrward:=TRUE;
	 		 ConveyorMotor.M_MoveBackward(); 
		  END_IF
		  
		tonTimeDelay.IN := NOT SensorOnConveyor;		
		IF tonTimeDelay.Q THEN
			tonTimeOut.IN := FALSE;
			uiExecutingStep:=2700;
		END_IF
		
		tonTimeOut.IN := TRUE;
	IF tonTimeOut.Q THEN
		tonTimeOut.IN := FALSE;
		_Abort :=TRUE;
		strStatus :='FB_OutRobot_RareBoxMove Step 2600: Move box out timeout';
	END_IF
2700: // Stop movor
		bMoveConveyorForward:=FALSE;
		bMoveConveyorBackrward:=FALSE;
		ConveyorMotor.M_MotorStop();
		tonTimeDelay.IN := FALSE;
		IF ConveyorMotor.InStopped THEN
			uiExecutingStep:=3000;
		END_IF
3000: // Finish	
	_Executed:=TRUE;
	
END_CASE
	
IF NOT Execute THEN
	eState:=STATE_RESETTING;
END_IF
IF _Error THEN
	eState:=STATE_ERROR;
END_IF
IF _Abort THEN
	eSTATE:=STATE_ABORTING;
END_IF
IF _Executed THEN
	eSTATE:=STATE_Done;
END_IF
END_METHOD

METHOD  M_STATE_RESETTING
VAR_INPUT
END_VAR
Error :=_Error;
Done :=_Executed;
Busy := FALSE;



CASE uiResettingStep OF
	
	0:
		ConveyorMotor.M_MotorStop();
		M_RecoveryAllObjects();
		uiResettingStep:=9999;


	9999:
		_ResetCompleted:=TRUE;
END_CASE
IF _ResetCompleted THEN
	eSTATE:=STATE_DORMANT;
END_IF
END_METHOD

END_FUNCTION_BLOCK

// ---- Library/20_MachineUnits/22_AllocateArea/Old_Version_Service/FB_PullOutConveyorAction_OLD.TcPOU
FUNCTION_BLOCK FB_PullOutConveyorAction_OLD EXTENDS FB_ObjectBase_V2 IMPLEMENTS IBasicElement
VAR_INPUT
    FixCylinderA1    : REFERENCE TO FB_Cylinder; // Conveyor A-side 1st cylinder
    FixCylinderA2    : REFERENCE TO FB_Cylinder; // Conveyor A-side 2nd cylinder
    FixCylinderB1    : REFERENCE TO FB_Cylinder; // Conveyor B-side 1st cylinder
    FixCylinderB2    : REFERENCE TO FB_Cylinder; // Conveyor B-side 2nd cylinder
    BarrierCylinderA : REFERENCE TO FB_Cylinder; // Conveyor A-side Barrier cylinder
    BarrierCylinderB : REFERENCE TO FB_Cylinder; // Conveyor B-side Barrier cylinder
    ConveyorMotorA    : REFERENCE TO FB_Motor; // PullOut Conveyor Motor 
	ConveyorMotorB	 : REFERENCE TO FB_Motor; //  Add New Motor Iomapping  edit Min 20250408
	INPUT            : REFERENCE TO ST_InputTable;	
    PullOutInfo      : ST_PullOutConveyorInfo;
END_VAR
VAR_OUTPUT
END_VAR
VAR
	FeedInSensor_A   : BOOL; // PullOut Conveyor A-side FeedIn Sensor
    FeedOutSensor_A  : BOOL; // PullOut Conveyor A-side FeedOut sensor
    DetactSensor_A   : BOOL; // PullOut Conveyor A-side detact sensor
    FeedInSensor_B   : BOOL; // PullOut Conveyor B-side FeedIn Sensor
    FeedOutSensor_B  : BOOL; // PullOut Conveyor B-side FeedOut sensor
    DetactSensor_B   : BOOL; // PullOut Conveyor B-side detact sensor
    TON_MotorRun     : TON; // Pull out conveyor motor running timer.
	TON_MotorReverse : TON; // Pull out conveyor motor reverse timer.
    TON_ForceForward : TON; // When auto process on, the time of force running in command direction.
	TON_MotorStopDelay : TON; // When Conveyor motor stop, the motor will be stopped later, so we need to give a time delay. 
    TON_BoxArrivedDelay: TON; // Check Box arrived(BoxA and BoxB) and delay.
	TON_BarryDelay : TON;
	tonFeedOutTimeOut :TON;
	tonMotorBReverse :TON;
	tonSensorDetectDelay : TON;
	TON_FeedInsensorADelay	:TON;
	TON_betweenboxReverse 	:TON;
	TON_PullOutTimeOut		:TON;
	//_Abort           : BOOL;
	bError			 : BOOL;
	strStatus	     : STRING;
	_UniqueErrorCode : STRING;
	PreviousStrStatus : STRING;
	PreviousErrorCode : STRING;
END_VAR

A00_BasicUnits();
A10_StateControl();

ACTION A00_BasicUnits:
TON_MotorRun		(PT	:= PullOutInfo.ConveyorRunningTime);
TON_MotorReverse	(PT	:= PullOutInfo.ConveyorReverseTime);
TON_ForceForward	(PT	:= T#0.5S);
TON_MotorStopDelay	(PT := PullOutInfo.ConveyorReverseTime);
TON_BoxArrivedDelay	(PT := T#800MS);
TON_BarryDelay		(PT	:= T#0.1S);
tonFeedOutTimeOut	(PT := PullOutInfo.ConveyorReverseTime*3 );		//notthing use
tonMotorBReverse	(PT := T#1.5S);


tonSensorDetectDelay(PT	:= T#100MS);
TON_FeedInsensorADelay(PT :=T#700MS);
TON_betweenboxReverse(PT :=T#700MS);
TON_PullOutTimeOut (PT :=T#20.0S);



ErrorID :=2750;
END_ACTION

ACTION A01_clcExecuting:
FeedInSensor_A  :=INPUT.bPullOutCV_AsideEntry_Sensor;
FeedOutSensor_A  :=INPUT.bPullOutCV_AsideExit_Sensor;
DetactSensor_A   :=input.bPullOutCV_Aside2ndBoxGap_Sensor;
FeedInSensor_B   :=INPUT.bPullOutCV_BsideEntry_Sensor;
FeedOutSensor_B  := INPUT.bPullOutCV_BsideExit_Sensor;
DetactSensor_B   := INPUT.bPullOutCV_Bside2ndBoxGap_Sensor;
END_ACTION

METHOD M_CheckCommand : BOOL
VAR_INPUT
END_VAR
M_CheckCommand := true;
END_METHOD

METHOD M_ResetCylinder : BOOL
VAR_INPUT
END_VAR
END_METHOD

METHOD  M_STATE_ABORTED
VAR_INPUT
END_VAR
uiAbortingStep := 0;
Busy := FALSE;
Aborted := TRUE;
_Abort := FALSE;
Error :=TRUE;
Status:= strStatus;
UniqueErrorCode:=_UniqueErrorCode;
IF NOT Execute THEN
		eState := STATE_RESETTING;
ELSIF reset AND Execute (*AND NOT error*) THEN
	
	CASE uiExecutingStep OF 
		50000:	//SlideA_FeedIn_Ext Resume step
				error :=FALSE;
				uiExecutingStep := 11000;	
	
	END_CASE
	eState := STATE_EXECUTING;
END_IF



//IF NOT Execute THEN
//	eState := STATE_RESETTING;
//ELSIF reset THEN
//	PreviousStrStatus := strStatus;
//	PreviousErrorCode := _UniqueErrorCode;
//	IF (uiExecutingStep = 1030) OR
//		(uiExecutingStep = 2030) OR
//		(uiExecutingStep = 3030)
// 	THEN
//		eState := STATE_EXECUTING;
//	END_IF
//END_IF
END_METHOD

METHOD  M_STATE_ABORTING
VAR_INPUT
END_VAR
CASE uiAbortingStep OF
	0:
		IF strStatus = PreviousStrStatus THEN
			_UniqueErrorCode :=PreviousErrorCode;
		END_IF
		TON_MotorRun.IN := FALSE;
		ConveyorMotorA.M_MotorStop();// .M_StopMotor('Aborting');
		TON_MotorStopDelay.IN := TRUE;
		uiAbortingStep := 100;
	100:
		_Abort :=FALSE;
		IF ConveyorMotorA.InStopped AND TON_MotorStopDelay.Q THEN
			uiAbortingStep := 200;
		END_IF
	200:
		TON_MotorStopDelay.IN := FALSE;
	//DAS.fbStorageArea.M_InactivePulloutConveyorInternCtrl();
		uiAbortingStep := 300;
	300:
		eState := STATE_Aborted;
END_CASE
END_METHOD

METHOD  M_STATE_DONE
VAR_INPUT
END_VAR
Busy := FALSE;
Done := TRUE;
//
IF NOT Execute THEN
	eState := STATE_RESETTING;
END_IF
END_METHOD

METHOD  M_STATE_DORMANT
VAR_INPUT
END_VAR
Busy    := FALSE;
Done    := FALSE;
Aborted := FALSE;
Error   := FALSE;
_Error :=FALSE;
ErrorID := 0;
Status  := '';
uiExecutingStep := 0;
uiResettingStep := 0;
uiAbortingStep :=0;
_Abort := FALSE;
_Executed := FALSE;
_ResetCompleted := FALSE;
TON_MotorRun.IN := FALSE;
TON_MotorReverse.IN := FALSE;
TON_ForceForward.IN := FALSE;
TON_MotorStopDelay.IN := FALSE;
TON_BoxArrivedDelay.IN := FALSE;
tonFeedOutTimeOut.IN :=FALSE;
tonMotorBReverse.IN :=FALSE;
tonSensorDetectDelay.IN:=FALSE;

TON_FeedInsensorADelay.IN :=FALSE;
TON_betweenboxReverse.IN :=FALSE;
TON_PullOutTimeOut.IN :=FALSE;
PreviousStrStatus			 :='';
PreviousErrorCode			 :='';
//DAS.fbStorageArea.M_InactivePulloutConveyorInternCtrl();
IF Execute THEN
	eState := STATE_EXECUTING;
END_IF
END_METHOD

METHOD  M_STATE_ERROR
VAR_INPUT
END_VAR

Status :=strStatus;
Error:=TRUE;
Busy :=FALSE;
Done :=FALSE;
UniqueErrorCode:=_UniqueErrorCode;
ConveyorMotorA.M_MotorStop();
ConveyorMotorB.M_MotorStop();
IF NOT Execute THEN
	eState :=STATE_RESETTING;
END_IF
END_METHOD

METHOD  M_STATE_EXECUTING
VAR_INPUT
END_VAR
VAR_INST	
END_VAR
Busy := TRUE;
A01_clcExecuting();
CASE uiExecutingStep OF
    0:
        IF M_CheckCommand() THEN
            uiExecutingStep := 100;
        ELSE
            Status := 'Wrong command, check the command setting';
            _Error := TRUE;
        END_IF
    100:
        FixCylinderA1.M_Retract();// .M_Retract();//('Clear command');
        FixCylinderA2.M_Retract();//('Clear command');
        FixCylinderB1.M_Retract();//('Clear command');
        FixCylinderB2.M_Retract();//('Clear command');
        BarrierCylinderA.M_Retract();//('Clear command');
        BarrierCylinderB.M_Retract();//('Clear command');

        IF FixCylinderA1.InRearPosition AND
           FixCylinderA2.InRearPosition AND
           FixCylinderB1.InRearPosition AND
           FixCylinderB2.InRearPosition AND
           BarrierCylinderA.InRearPosition AND
           BarrierCylinderB.InRearPosition THEN
            uiExecutingStep := 500;
        END_IF
    500:
        CASE PullOutInfo.CommandType OF
            E_PullOutConveyorCommandType.SideA_FeedIn:
                uiExecutingStep := 1000;
            E_PullOutConveyorCommandType.SideB_FeedIn:
                uiExecutingStep := 2000;
            E_PullOutConveyorCommandType.Both_FeedIn:
                uiExecutingStep := 3000;
            E_PullOutConveyorCommandType.SideA_FeedOut:
                uiExecutingStep := 4000;
            E_PullOutConveyorCommandType.SideB_FeedOut:
                uiExecutingStep := 5000;
            E_PullOutConveyorCommandType.Both_FeedOut:
                uiExecutingStep := 6000;
            E_PullOutConveyorCommandType.MoveForward:
                uiExecutingStep := 7000;
            E_PullOutConveyorCommandType.MoveBackward:
                uiExecutingStep := 8000;
			E_PullOutConveyorCommandType.SlideA_FeedOut_Ext:
				uiExecutingStep := 9000;
			E_PullOutConveyorCommandType.SlideB_FeedOut_Ext:
				uiExecutingStep := 10000;
			E_PullOutConveyorCommandType.SlideA_FeedIn_Ext:
				uiExecutingStep := 11000;
			E_PullOutConveyorCommandType.SlideB_FeedIn_Ext:
				uiExecutingStep := 12000;
        ELSE
            Status := 'Command type out of range.';
            _Error := TRUE;
        END_CASE
		
{region "SideA_FeedIn"}
    1000:
        // Side A feed in box start.
        TON_ForceForward.IN := TRUE;
        ConveyorMotorA.M_MoveForward();// .M_Extend();//;// .M_Extend();//;//('Force forward');

        IF TON_ForceForward.Q THEN
            uiExecutingStep := 1010;
        END_IF
    1010:
        TON_ForceForward.IN := FALSE;
        ConveyorMotorA.M_MotorStop();// .M_MotorStop();//('Force forward stop');
        TON_MotorStopDelay.IN := TRUE;

        IF ConveyorMotorA.InStopped  AND TON_MotorStopDelay.Q THEN
            uiExecutingStep := 1020;
        END_IF
    1020:
        TON_MotorStopDelay.IN := FALSE;
		TON_BoxArrivedDelay.IN := FeedInSensor_A;
        IF TON_BoxArrivedDelay.Q THEN
            uiExecutingStep := 1100;
        ELSE
			TON_BoxArrivedDelay.IN := FALSE;
            uiExecutingStep := 1030;
        END_IF
    1030:
		TON_BoxArrivedDelay.IN := FeedInSensor_A;
        ConveyorMotorA.M_MoveForward();// .M_Extend();//;//('');
        TON_MotorRun.IN := TRUE;

        IF TON_BoxArrivedDelay.Q THEN
            uiExecutingStep := 1100;
        ELSIF TON_MotorRun.Q THEN
            Status := 'SideA FeedIn no box.';
            _Abort := TRUE;
        END_IF
    1100:
        TON_MotorRun.IN       := FALSE;
        TON_MotorStopDelay.IN := TRUE;
        ConveyorMotorA.M_MotorStop();//('');

        IF ConveyorMotorA.InStopped  AND TON_MotorStopDelay.Q THEN
            uiExecutingStep := 1200;
        END_IF
    1200:
        TON_MotorStopDelay.IN := FALSE;
        FixCylinderA1.M_Extend();// .M_Extend();//('');

        IF FixCylinderA1.InFrontPosition THEN
            uiExecutingStep := 1300;
        END_IF
    1300:
        ConveyorMotorA.M_MoveBackward();// .M_MoveBackward();//('');
        TON_MotorReverse.IN := TRUE;

        IF TON_MotorReverse.Q THEN
            uiExecutingStep := 1400;
        END_IF
    1400:
        ConveyorMotorA.M_MotorStop();//('');
        TON_MotorReverse.IN   := FALSE;
        TON_MotorStopDelay.IN := TRUE;

        IF ConveyorMotorA.InStopped  AND TON_MotorStopDelay.Q THEN
            uiExecutingStep := 1500;
        END_IF
    1500:
        TON_MotorStopDelay.IN := FALSE;
        FixCylinderA1.M_Retract();//('');

        IF FixCylinderA1.InRearPosition THEN
            uiExecutingStep := 99000;
        END_IF

{endregion}

{region "SideB_FeedIn"}
 2000:
        // Side-B feed in start
        TON_ForceForward.IN := TRUE;
        ConveyorMotorB.M_MoveForward(); //('Force forward');

        IF TON_ForceForward.Q THEN
            uiExecutingStep := 2010;
        END_IF
    2010:
        TON_ForceForward.IN   := FALSE;
        TON_MotorStopDelay.IN := TRUE;
        ConveyorMotorB.M_MotorStop();//('Force forward stop');

        IF ConveyorMotorA.InStopped  AND TON_MotorStopDelay.Q THEN
            uiExecutingStep := 2020;
        END_IF
    2020:
        TON_MotorStopDelay.IN := FALSE;
		TON_BoxArrivedDelay.IN := FeedInSensor_B;
        IF TON_BoxArrivedDelay.Q THEN
            uiExecutingStep := 2100;
        ELSE
			TON_BoxArrivedDelay.IN := FALSE;
            uiExecutingStep := 2030;
        END_IF
    2030:
        ConveyorMotorB.M_MoveForward();// 
        TON_MotorRun.IN := TRUE;
		TON_BoxArrivedDelay.IN := FeedInSensor_B;
        IF TON_BoxArrivedDelay.Q THEN
            uiExecutingStep := 2100;
        ELSIF TON_MotorRun.Q THEN
            Status := 'SideB FeedIn no box.';
            _Abort := TRUE;
        END_IF
    2100:
        TON_MotorRun.IN       := FALSE;
        TON_MotorStopDelay.IN := TRUE;
        ConveyorMotorB.M_MotorStop();//('');

        IF ConveyorMotorB.InStopped  AND TON_MotorStopDelay.Q THEN
            uiExecutingStep := 2200;
        END_IF
    2200:
        TON_MotorStopDelay.IN := FALSE;
        FixCylinderB1.M_Extend();//('');

        IF FixCylinderB1.InFrontPosition THEN
            uiExecutingStep := 2300;
        END_IF
    2300:
        ConveyorMotorB.M_MoveBackward();//('');
        TON_MotorReverse.IN := TRUE;

        IF TON_MotorReverse.Q THEN
            uiExecutingStep := 2400;
        END_IF
    2400:
        ConveyorMotorB.M_MotorStop();//('');
        TON_MotorReverse.IN   := FALSE;
        TON_MotorStopDelay.IN := TRUE;

        IF ConveyorMotorB.InStopped  AND TON_MotorStopDelay.Q THEN
            uiExecutingStep := 2500;
        END_IF
    2500:
        TON_MotorStopDelay.IN := FALSE;
        FixCylinderB1.M_Retract();//('');

        IF FixCylinderB1.InRearPosition THEN
            uiExecutingStep := 99000;
        END_IF
{endregion}

{region "Both_FeedIn"}

    3000:
        // Both side feed in start
        TON_ForceForward.IN := TRUE;
        ConveyorMotorA.M_MoveForward();// ('Force forward');
		ConveyorMotorB.M_MoveForward();// 

        IF TON_ForceForward.Q THEN
            uiExecutingStep := 3010;
        END_IF
    3010:
        TON_ForceForward.IN   := FALSE;
        TON_MotorStopDelay.IN := TRUE;
        ConveyorMotorA.M_MotorStop();//('Force forward stop');
		ConveyorMotorB.M_MotorStop();//('Force forward stop');
		
        IF ConveyorMotorA.InStopped  AND ConveyorMotorB.InStopped  AND TON_MotorStopDelay.Q THEN
            uiExecutingStep := 3020;
        END_IF
    3020:
        TON_MotorStopDelay.IN := FALSE;
		ConveyorMotorA.M_MoveForward();//('Force forward');
		ConveyorMotorB.M_MoveForward();//;//('Force forward');
		
		TON_BoxArrivedDelay.IN := FeedInSensor_A AND FeedInSensor_B;
        IF TON_BoxArrivedDelay.Q THEN
            uiExecutingStep := 3100;
        ELSE
			TON_BoxArrivedDelay.IN := FALSE;
            uiExecutingStep := 3030;
        END_IF
    3030:
        ConveyorMotorA.M_MoveForward();//;//('');
		ConveyorMotorB.M_MoveForward();//;//('');
        TON_MotorRun.IN := TRUE;
		TON_BoxArrivedDelay.IN := FeedInSensor_A AND FeedInSensor_B;
        IF  TON_BoxArrivedDelay.Q THEN
            uiExecutingStep := 3100;
        ELSIF TON_MotorRun.Q THEN
            Status := 'SideA or SideB FeedIn no box.';
            _Abort := TRUE;
        END_IF
    3100:
        TON_MotorRun.IN       := FALSE;
        TON_MotorStopDelay.IN := TRUE;
        ConveyorMotorA.M_MotorStop();//('');
		ConveyorMotorB.M_MotorStop();//('');
		

        IF ConveyorMotorA.InStopped  AND ConveyorMotorB.InStopped  AND TON_MotorStopDelay.Q THEN
            uiExecutingStep := 3200;
        END_IF
    3200:
        TON_MotorStopDelay.IN := FALSE;
        FixCylinderB1.M_Extend();//('');
        FixCylinderA1.M_Extend();//('');

        IF FixCylinderA1.InFrontPosition AND FixCylinderB1.InFrontPosition THEN
            uiExecutingStep := 3300;
        END_IF
    3300:
        ConveyorMotorA.M_MoveBackward();//('');
		ConveyorMotorB.M_MoveBackward();//('');
        TON_MotorReverse.IN := TRUE;

        IF TON_MotorReverse.Q THEN
            uiExecutingStep := 3400;
        END_IF
    3400:
        ConveyorMotorA.M_MotorStop();//('');
		ConveyorMotorB.M_MotorStop();//('');
        TON_MotorReverse.IN   := FALSE;
        TON_MotorStopDelay.IN := TRUE;

        IF ConveyorMotorA.InStopped  AND ConveyorMotorB.InStopped  AND TON_MotorStopDelay.Q THEN
            uiExecutingStep := 3500;
        END_IF
    3500:
        FixCylinderA1.M_Retract();//('');
        FixCylinderB1.M_Retract();//('');

        IF FixCylinderA1.InRearPosition AND FixCylinderB1.InRearPosition THEN
            uiExecutingStep := 99000;
        END_IF			 
{endregion}

{region "SideA_FeedOut"}
    4000:	//SideA_FeedOut
        ConveyorMotorA.M_MoveBackward();//('');
        TON_MotorReverse.IN := TRUE;

        IF TON_MotorReverse.Q AND NOT FeedInSensor_A THEN
            uiExecutingStep := 4500;
        END_IF
    4500:
        ConveyorMotorA.M_MotorStop();//('');
        TON_MotorReverse.IN   := FALSE;
        TON_MotorStopDelay.IN := TRUE;

        IF ConveyorMotorA.InStopped  AND TON_MotorStopDelay.Q THEN
            uiExecutingStep := 99000;
        END_IF
{endregion}

{region "SideB_FeedOut"}
    5000:	//SideB_FeedOut
        ConveyorMotorB.M_MoveBackward();//('');
        TON_MotorReverse.IN   := TRUE;
        TON_MotorStopDelay.IN := FALSE;

        IF TON_MotorReverse.Q AND NOT FeedInSensor_B THEN
            uiExecutingStep := 5500;
        END_IF
    5500:
        ConveyorMotorB.M_MotorStop();//('');
        TON_MotorReverse.IN   := FALSE;
        TON_MotorStopDelay.IN := TRUE;

        IF ConveyorMotorB.InStopped  AND TON_MotorStopDelay.Q THEN
            uiExecutingStep := 99000;
        END_IF
{endregion}

{region "Both_FeedOut"}
    6000:	//Both_FeedOut
        ConveyorMotorA.M_MoveBackward();//('');
		ConveyorMotorB.M_MoveBackward();//('');
        TON_MotorReverse.IN   := TRUE;
        TON_MotorStopDelay.IN := FALSE;

        IF TON_MotorReverse.Q AND NOT FeedInSensor_A AND NOT FeedInSensor_B THEN
            uiExecutingStep := 6500;
        END_IF
    6500:
        ConveyorMotorA.M_MotorStop();//('');
		ConveyorMotorB.M_MotorStop();//('');
        TON_MotorReverse.IN   := FALSE;
        TON_MotorStopDelay.IN := TRUE;

        IF ConveyorMotorA.InStopped  AND ConveyorMotorB.InStopped  AND TON_MotorStopDelay.Q THEN
            uiExecutingStep := 99000;
        END_IF			 
{endregion}

{region "MoveForward"}
    7000:
        // Move forward start
        ConveyorMotorA.M_MoveForward();//;//('Move forward');
		ConveyorMotorB.M_MoveForward();//;//('Move forward');
        TON_MotorRun.IN := TRUE;
        uiExecutingStep := 7100;
    7100:
        IF TON_MotorRun.Q THEN
            ConveyorMotorA.M_MotorStop();//('Stop');
			ConveyorMotorB.M_MotorStop();//('Stop');
            uiExecutingStep := 7200;
        END_IF
    7200:
        TON_MotorRun.IN       := FALSE;
        TON_MotorStopDelay.IN := TRUE;

        IF ConveyorMotorA.InStopped  AND ConveyorMotorB.InStopped  AND TON_MotorStopDelay.Q THEN
            uiExecutingStep := 99000;
        END_IF
{endregion}

{region "MoveBackward"}
    8000:
        // Move backward start
        ConveyorMotorA.M_MoveBackward();//('Move backward');
		ConveyorMotorB.M_MoveBackward();//('Move backward');
        TON_MotorReverse.IN := TRUE;
        uiExecutingStep := 8100;
    8100:
        IF TON_MotorReverse.Q THEN
            ConveyorMotorA.M_MotorStop();//('Stop');
			ConveyorMotorB.M_MotorStop();//('Stop');
            uiExecutingStep := 8200;
        END_IF
    8200:
        TON_MotorRun.IN       := FALSE;
        TON_MotorStopDelay.IN := TRUE;

        IF ConveyorMotorA.InStopped  AND ConveyorMotorB.InStopped  AND TON_MotorStopDelay.Q THEN
            uiExecutingStep := 99000;
        END_IF 
{endregion}

{region "SlideA_FeedOut_Ext"}
//	9000: // SlideA_FeedOut_Ext
//		ConveyorMotor.M_MoveBackward();//('');
//		TON_BoxArrivedDelay.IN := TRUE;
//		IF NOT FeedInSensor_A THEN
//			TON_MotorStopDelay.IN := TRUE;
//			IF TON_MotorStopDelay.Q THEN
//				ConveyorMotor.M_MotorStop();//('');
//				TON_BoxArrivedDelay.IN := FALSE;
//				uiExecutingStep := 99000;
//			END_IF
//		END_IF
//		IF TON_BoxArrivedDelay.Q THEN
//			Status := 'SlideA box is still there';
//			_Error := TRUE;
//		END_IF
	9000: //SlideA FeedOut_Ext
			ConveyorMotorA.M_MoveBackward();//('');
			tonMotorBReverse.IN :=TRUE;
			IF tonMotorBReverse.Q THEN
				ConveyorMotorA.M_MotorStop();//('');
				uiExecutingStep :=9100;
			END_IF
	9100:	//check sensor make sure full box behide
			IF ConveyorMotorA.InStopped  THEN
				IF (NOT FeedInSensor_A) AND 
					(NOT DetactSensor_A) THEN
					uiExecutingStep :=99000;
				ELSIF FeedInSensor_A OR
						DetactSensor_A THEN
						_Error :=TRUE;
						strStatus :='PullOutConveyorA FeedOut full box ,please remove ';
				END_IF
			END_IF
{endregion}

{region "SlideB_FeedOut_Ext"}
//	10000: // SlideB_FeedOut_Ext
	
//		ConveyorMotorB.M_MoveBackward();//('');
//		TON_BoxArrivedDelay.IN := TRUE;
//		IF NOT FeedInSensor_B THEN
//			TON_MotorStopDelay.IN := TRUE;
//			IF TON_MotorStopDelay.Q THEN
//				ConveyorMotorB.M_MotorStop();//('');
//				TON_BoxArrivedDelay.IN := FALSE;
//				uiExecutingStep := 99000;
//			END_IF
//		END_IF
//		IF TON_BoxArrivedDelay.Q THEN
//			Status := 'SlideB box is still there';
//			_Error := TRUE;
//		END_IF

	//======================	SlideA FeedOut_Ext
	10000: 
			ConveyorMotorB.M_MoveBackward();//('');
			tonMotorBReverse.IN :=TRUE;
			IF tonMotorBReverse.Q THEN
				ConveyorMotorB.M_MotorStop();//('');
				uiExecutingStep :=10100;
			END_IF
	10100:	//check sensor make sure full box behide
			IF ConveyorMotorB.InStopped  THEN
				IF (NOT FeedInSensor_B) AND 
					(NOT DetactSensor_B) THEN
					uiExecutingStep :=99000;
				ELSIF FeedInSensor_B OR
						DetactSensor_B THEN
						_Error :=TRUE;
						strStatus :='PullOutConveyorB FeedOut full box ,please remove ';
				END_IF
			END_IF
{endregion}

{region "SlideA_FeedIn_Ext"}
	//=======================	SlideA_FeedIn_Ext	near storage side
	11000: 
		IF 	DetactSensor_A AND FeedInSensor_A THEN
			uiExecutingStep := 11100;
		ELSIF NOT DetactSensor_A AND FeedInSensor_A THEN
			uiExecutingStep := 11200;
		ELSIF DetactSensor_A AND NOT FeedInSensor_A THEN
			uiExecutingStep := 11400;
		ELSIF NOT DetactSensor_A AND NOT FeedInSensor_A THEN
			uiExecutingStep := 11400;
		END_IF
	11100: 	// two sensor on
			// Reversemotor unstill two sensor off
		ConveyorMotorA.M_MoveBackward();//('');
		tonMotorBReverse.IN :=TRUE;
		IF tonMotorBReverse.Q THEN
			tonMotorBReverse.IN :=FALSE;
			ConveyorMotorA.M_MotorStop();//('');
			uiExecutingStep :=11110;
		END_IF
		
	11110:	//wait conveyorA stop
		IF ConveyorMotorA.InStopped  THEN
			uiExecutingStep :=11120;
		END_IF
	11120:	//check two sensor
		IF DetactSensor_A OR FeedInSensor_A THEN
			//_Error :=TRUE;
			strStatus :='PullOutConveyorA full box ,please remove';
			uiExecutingStep :=50000;	//abort step
		ELSE 
			uiExecutingStep :=11800;
		END_IF
		
	11200:	// FeedinSensor on
			//conveyor forward 
			FixCylinderA2.M_Extend();//('');
			IF  FixCylinderA2.InFrontPosition THEN
				ConveyorMotorA.M_MoveForward();// .M_Extend();//;//('');
				uiExecutingStep := 11840;
			END_IF		
	
	11400:	//two sensor off , need make sure no box in two sensor between 
			// Reverse motor to touch detactSensor , make sure no box 
			ConveyorMotorA.M_MoveBackward();//('');
			TON_betweenboxReverse.IN :=TRUE;
			IF TON_betweenboxReverse.Q THEN
				TON_betweenboxReverse.IN :=FALSE;
				ConveyorMotorA.M_MotorStop();//('');
				uiExecutingStep := 11410;
			END_IF
	11410:
			// wait motor stop
			IF ConveyorMotorA.InStopped  THEN
				uiExecutingStep :=11420;
			END_IF
	11420:	//check sensor
			IF DetactSensor_A THEN
				uiExecutingStep :=11430; // todo sth
			ELSIF NOT DetactSensor_A  THEN
				uiExecutingStep :=11800;
			END_IF 
	11430:	//reversemotor unstill sensor off
			ConveyorMotorA.M_MoveBackward();//('');
			TON_betweenboxReverse.IN :=TRUE;	//use to timeout 0.6s
			IF NOT DetactSensor_A THEN
				ConveyorMotorA.M_MotorStop();//('');
				uiExecutingStep :=11440;
			END_IF
			IF TON_betweenboxReverse.Q THEN
				//_Error :=TRUE;
				strStatus :='PullOutConveyorA FeedIn full box ,please remove box';
				uiExecutingStep :=50000;
			END_IF
	11440:	//wait motor stop
			IF ConveyorMotorA.InStopped  THEN
				uiExecutingStep :=11800;
			END_IF
			
	11800:	//BlockA forward and motorA forward
			BarrierCylinderA.M_Extend();//('');
			IF BarrierCylinderA.InFrontPosition THEN
				ConveyorMotorA.M_MoveForward();//;//('');
				uiExecutingStep :=11810;
			END_IF
	11810:	//wait box move in sensor and pressbox forward
			TON_PullOutTimeOut.IN 	:=TRUE;		//10S
			tonSensorDetectDelay.IN :=DetactSensor_A;		//100MS
			IF tonSensorDetectDelay.Q THEN
				tonSensorDetectDelay.IN :=FALSE;
				TON_PullOutTimeOut.IN 	:=FALSE;
				FixCylinderA2.M_Extend();//('');
				uiExecutingStep :=11820;
			END_IF
			IF TON_PullOutTimeOut.Q THEN
				//_Error :=TRUE;
				strStatus :='PullOutConveyorA none box ,please refill box';
				uiExecutingStep := 50000;
			END_IF
	11820:	//wait PressboxA2 forward and Blockbox backward 
			IF FixCylinderA2.InFrontPosition THEN
				BarrierCylinderA.M_Retract();//('');
				uiExecutingStep :=11830;
			END_IF
	11830:	//wait blockbox backward
			IF BarrierCylinderA.InRearPosition THEN
				uiExecutingStep :=11840;
			END_IF
	11840:	//delay sensor time
			TON_FeedInsensorADelay.IN := FeedInSensor_A ;
			IF TON_FeedInsensorADelay.Q THEN
				TON_FeedInsensorADelay.IN :=FALSE;
				ConveyorMotorA.M_MotorStop();//('');
				uiExecutingStep :=11850;
			END_IF
	11850:	//wait conveyor stop
			IF ConveyorMotorA.InStopped  THEN
				FixCylinderA1.M_Extend();//('');
				uiExecutingStep :=11860;
			END_IF
	11860:	//wait pressbox cylinder move
			IF FixCylinderA1.InFrontPosition THEN
				FixCylinderA1.M_Retract();//('');
				FixCylinderA2.M_Retract();//('');
				uiExecutingStep :=11870;
			END_IF
	11870:	//done
			IF FixCylinderA1.InRearPosition AND FixCylinderA2.InRearPosition THEN
				uiExecutingStep :=99000;
			END_IF
//	11100:
//		// SlideA has two box in the front position
//		// Fix the frontmost box
//		FixCylinderA1.M_Extend();//('');
//		IF FixCylinderA1.InFrontPosition THEN
//			uiExecutingStep := 11110;
//		END_IF
//	11110:
//		// PulloutConveyor reverse to separate two boxes
//		ConveyorMotor.M_MoveBackward();//('');
//		TON_BoxArrivedDelay.IN := TRUE;
//		IF TON_BoxArrivedDelay.Q OR NOT DetactSensor_A THEN
//			uiExecutingStep := 11120;
//		END_IF
//	11120:
//		ConveyorMotor.M_MotorStop();//('');
//		TON_MotorStopDelay.IN := TRUE;
//		IF TON_MotorStopDelay.Q THEN
//			uiExecutingStep := 11130;
//		END_IF
//	11130:
//		FixCylinderA1.M_Retract();//('');
//		IF FixCylinderA1.InRearPosition// THEN
//			uiExecutingStep := 99000;
//		END_IF
//	11200:
//		// SlidA has a box in the front position, and not detact then second box
//		BarrierCylinderA.M_Extend();//('');
//		IF BarrierCylinderA.In_FrontPosition THEN
//			uiExecutingStep := 11210;
//		END_IF
//	11210:
//		// Check the front box arrived
//		ConveyorMotor.M_Extend();//;//('');
//		TON_BoxArrivedDelay.IN := TRUE;
//		IF TON_BoxArrivedDelay.Q THEN
//			uiExecutingStep := 11220;
//		END_IF
//	11220:
//		ConveyorMotor.M_MotorStop();//('');
//		TON_MotorStopDelay.IN := TRUE;
//		IF TON_MotorStopDelay.Q THEN
//			uiExecutingStep := 11230;
//		END_IF
//	11230:
//		FixCylinderA1.M_Extend();//('');
//		IF FixCylinderA1.InFrontPosition THEN
//			uiExecutingStep := 11240;
//		END_IF
//	11240:
//		FixCylinderA1.M_Retract();//('');
//		IF FixCylinderA1.InRearPosition// THEN
//			uiExecutingStep := 99000;
//		END_IF
//	11400:
//		// SlideA has no boxex in the front position
//		// Rise the barrier
//		BarrierCylinderA.M_Extend();//('');
//		IF BarrierCylinderA.In_FrontPosition THEN
//			uiExecutingStep := 11410;
//		END_IF
//	11410:
//		ConveyorMotor.M_Extend();//;//('');
		
//		IF DetactSensor_A THEN
//			uiExecutingStep := 11420;
//		END_IF
////		IF TON_BoxArrivedDelay.Q THEN
////			Status:= 'SlideA FeedIn error';
////			_Error := TRUE;
////		END_IF
//	11420:
//		FixCylinderA2.M_Extend();//('');
//		TON_BoxArrivedDelay.IN := FALSE;
//		uiExecutingStep := 11430;
//	11430:
//		BarrierCylinderA.M_Retract();//('');
//		IF BarrierCylinderA.In_RearPosition THEN
//			uiExecutingStep := 11440;
//		END_IF
//	11440:
//		TON_BoxArrivedDelay.IN := TRUE;
//		IF FeedInSensor_A AND TON_BoxArrivedDelay.Q THEN
//			ConveyorMotor.M_MotorStop();//('');
//			uiExecutingStep := 11450;
//		END_IF
////		IF TON_BoxArrivedDelay.Q THEN
////			Status := 'SlideA FeedIn no box';
////			_Error := TRUE;
////		END_IF
//	11450:
//		FixCylinderA1.M_Extend();//('');
//		//TON_BoxArrivedDelay.IN := TRUE;
//		IF FixCylinderA1.InFrontPosition  THEN
//			uiExecutingStep := 11460;
//		END_IF
//	11460:
//		TON_BarryDelay.IN := TRUE;
//		IF TON_BarryDelay.Q THEN
//			FixCylinderA1.M_Retract();//('');
//			FixCylinderA2.M_Retract();//('');
//			uiExecutingStep := 99000;
//		END_IF
{endregion}

{region "SlideB_FeedIn_Ext"}
	//===========================	SlideB_FeedIn_Ext

	12000: 
		IF 	DetactSensor_B  AND FeedInSensor_B THEN
			uiExecutingStep := 12100;
		ELSIF NOT DetactSensor_B  AND FeedInSensor_B THEN
			uiExecutingStep := 12200;
		ELSIF DetactSensor_B  AND NOT FeedInSensor_B THEN
			uiExecutingStep := 12400;
		ELSIF NOT DetactSensor_B  AND NOT FeedInSensor_B THEN
			uiExecutingStep := 12400;
		END_IF
	12100: 	// two sensor on
			// Reversemotor unstill two sensor off
		ConveyorMotorB.M_MoveBackward();//('');
		tonMotorBReverse.IN :=TRUE;
		IF tonMotorBReverse.Q THEN
			tonMotorBReverse.IN :=FALSE;
			ConveyorMotorB.M_MotorStop();//('');
			uiExecutingStep :=12110;
		END_IF
		
	12110:	//wait conveyorA stop
		IF ConveyorMotorB.InStopped  THEN
			uiExecutingStep :=12120;
		END_IF
	12120:	//check two sensor
		IF DetactSensor_B OR FeedInSensor_B THEN
			_Error :=TRUE;
			strStatus :='PullOutConveyorB full box ,please remove';
		ELSE 
			uiExecutingStep :=12800;
		END_IF
		
	12200:	// FeedinSensor on
			//conveyor forward 
			FixCylinderB2.M_Extend();//('');
			IF  FixCylinderB2.InFrontPosition THEN
				ConveyorMotorB.M_MoveForward();// .M_Extend();//;//('');
				uiExecutingStep := 12840;
			END_IF		
	
	12400:	//two sensor off , need make sure no box in two sensor between 
			// Reverse motor to touch detactSensor , make sure no box 
			ConveyorMotorB.M_MoveBackward();//('');
			TON_betweenboxReverse.IN :=TRUE;
			IF TON_betweenboxReverse.Q THEN
				TON_betweenboxReverse.IN :=FALSE;
				ConveyorMotorB.M_MotorStop();//('');
				uiExecutingStep := 12410;
			END_IF
	12410:
			// wait motor stop
			IF ConveyorMotorB.InStopped  THEN
				uiExecutingStep :=12420;
			END_IF
	12420:	//check sensor
			IF DetactSensor_B THEN
				uiExecutingStep :=12430; // todo sth
			ELSIF NOT DetactSensor_B  THEN
				uiExecutingStep :=12800;
			END_IF 
	12430:	//reversemotor unstill sensor off
			ConveyorMotorB.M_MoveBackward();//('');
			TON_betweenboxReverse.IN :=TRUE;	//use to timeout 0.6s
			IF NOT DetactSensor_B THEN
				ConveyorMotorB.M_MotorStop();//('');
				uiExecutingStep :=12440;
			END_IF
			IF TON_betweenboxReverse.Q THEN
				_Error :=TRUE;
				strStatus :='PullOutConveyorB FeedIn full box ,please remove box';
			END_IF
	12440:	//wait motor stop
			IF ConveyorMotorB.InStopped  THEN
				uiExecutingStep :=12800;
			END_IF
			
	12800:	//BlockA forward and motorA forward
			BarrierCylinderB.M_Extend();//('');
			IF BarrierCylinderB.InFrontPosition THEN
				ConveyorMotorB.M_MoveForward();//;//('');
				uiExecutingStep :=12810;
			END_IF
	12810:	//wait box move in sensor and pressbox forward
			TON_PullOutTimeOut.IN 	:=TRUE;		//10S
			tonSensorDetectDelay.IN :=DetactSensor_B;		//100MS
			IF tonSensorDetectDelay.Q THEN
				tonSensorDetectDelay.IN :=FALSE;
				TON_PullOutTimeOut.IN 	:=FALSE;
				FixCylinderB2.M_Extend();//('');
				uiExecutingStep :=12820;
			END_IF
			IF TON_PullOutTimeOut.Q THEN
				_Error :=TRUE;
				strStatus :='PullOutConveyorA none box ,please refill box';
			END_IF
	12820:	//wait PressboxB2 forward & Blockbox backward 
			IF FixCylinderB2.InFrontPosition THEN
				BarrierCylinderB.M_Retract();//('');
				uiExecutingStep :=12830;
			END_IF
	12830:	//wait blockbox backward
			IF BarrierCylinderB.InRearPosition THEN
				uiExecutingStep :=12840;
			END_IF
	12840:	//delay sensor time
			TON_FeedInsensorADelay.IN := FeedInSensor_B ;
			IF TON_FeedInsensorADelay.Q THEN
				TON_FeedInsensorADelay.IN :=FALSE;
				ConveyorMotorB.M_MotorStop();//('');
				uiExecutingStep :=12850;
			END_IF
	12850:	//wait conveyor stop
			IF ConveyorMotorB.InStopped  THEN
				FixCylinderB1.M_Extend();//('');
				uiExecutingStep :=12860;
			END_IF
	12860:	//wait pressbox cylinder move
			IF FixCylinderB1.InFrontPosition THEN
				FixCylinderB1.M_Retract();//('');
				FixCylinderB2.M_Retract();//('');
				uiExecutingStep :=12870;
			END_IF
	12870:	//done
			IF FixCylinderB1.InRearPosition AND FixCylinderB2.InRearPosition THEN
				uiExecutingStep :=99000;
			END_IF
//	12000: 	
//			//check FeedinSensor & DetactSensor
//			tonMotorBReverse.IN :=TRUE;
//			ConveyorMotorb.M_MoveBackward();//('');				
//			IF tonMotorBReverse.Q  THEN
//					tonMotorBReverse.IN :=FALSE;
//					ConveyorMotorb.M_MotorStop();//('');
//					uiExecutingStep :=12005;
//			END_IF
//	12005: 	//check box leave sensor 
//			IF FeedInSensor_B OR DetactSensor_B THEN
//				_Error :=TRUE;
//				strStatus :='PullOutConveyorB full box ,please remove box';
//			ELSE
//				uiExecutingStep :=12010;
//			END_IF
	
//	12010:	//wait conveyorB stop
//			IF ConveyorMotorB.InStopped  THEN
//				uiExecutingStep := 12050;
//			END_IF
//	12050: 
//			//block forward 
//		BarrierCylinderB.M_Extend();//('');
//		IF BarrierCylinderB.In_FrontPosition THEN
//			uiExecutingStep := 12100;
//		END_IF
//	12100:	// motor forward & check detactsensor
//		ConveyorMotorB.M_Extend();//;//('');
//		TON_BoxArrivedDelay.IN := TRUE;
//		IF DetactSensor_B  THEN
//			uiExecutingStep := 12200;
//		END_IF
//		IF TON_BoxArrivedDelay.Q THEN
//			Status := 'SlideB FeedIn no box';
//			_Error := TRUE;
//		END_IF
//	12200:
//		tonSensorDetectDelay.IN :=TRUE;
//		IF tonSensorDetectDelay.Q THEN
//			FixCylinderB2.M_Extend();//('');
//			uiExecutingStep := 12300;
//		END_IF
//	12300:
//		tonSensorDetectDelay.IN :=FALSE;
//		BarrierCylinderB.M_Retract();//('');
//		IF BarrierCylinderB.In_RearPosition THEN
//			uiExecutingStep := 12400;
//		END_IF
//	12400:
//		TON_BoxArrivedDelay.IN := TRUE;
//		IF FeedInSensor_B THEN
//			ConveyorMotorB.M_MotorStop();//('');
//			uiExecutingStep := 12500;
//		END_IF
//		IF TON_BoxArrivedDelay.Q THEN
//			Status := 'SlideB FeedIn no box';
//			_Error := TRUE;
//		END_IF
//	12500:
//		FixCylinderB1.M_Extend();//('');
//		uiExecutingStep := 12510;
//	12510:
//		TON_BarryDelay.IN := TRUE;
//		IF TON_BarryDelay.Q THEN
//			FixCylinderB1.M_Retract();//('');
//			FixCylinderB2.M_Retract();//('');
//			uiExecutingStep := 99000;
//		END_IF
{endregion}

	50000:	//SlideA FeedIn Ext Resume step
			FixCylinderA1.M_Retract();
			FixCylinderA2.M_Retract();
			BarrierCylinderA.M_Retract();
			ConveyorMotorA.M_MotorStop();
			TON_PullOutTimeOut.IN :=FALSE;
			TON_betweenboxReverse.IN :=FALSE;
			IF FixCylinderA1.InRearPosition AND 
				FixCylinderA2.InRearPosition AND 
				BarrierCylinderA.InRearPosition AND 
				ConveyorMotorA.InStopped THEN
				_Abort :=TRUE;
			END_IF
			
    99000:
        TON_MotorStopDelay.IN := FALSE;
        _Executed             := TRUE;

END_CASE

IF _Executed THEN
    eState := STATE_DONE;
ELSIF NOT Execute THEN
    eState := STATE_RESETTING;
ELSIF _Abort OR Abort THEN
    eState := STATE_ABORTING;
ELSIF _Error THEN
	eState:=STATE_ERROR;	
END_IF
END_METHOD

METHOD  M_STATE_RESETTING
VAR_INPUT
END_VAR
CASE uiResettingStep OF
	0:
		FixCylinderA1.M_Retract();// .M_Retract();//('Resetting');
		FixCylinderA2.M_Retract();//('Resetting');
		FixCylinderB1.M_Retract();//('Resetting');
		FixCylinderB2.M_Retract();//('Resetting');
		BarrierCylinderA.M_Retract();//('Resetting');
		BarrierCylinderB.M_Retract();//('Resetting');
		uiResettingStep := 100;
	100:
		IF FixCylinderA1.InRearPosition AND
			FixCylinderA2.InRearPosition AND
			FixCylinderB1.InRearPosition AND
			FixCylinderB2.InRearPosition AND
			BarrierCylinderA.InRearPosition AND 
			BarrierCylinderB.InRearPosition THEN
			uiResettingStep := 200;
		END_IF
	200:
		ConveyorMotorA.M_MotorStop();// .M_StopMotor('Resetting');
		ConveyorMotorB.M_MotorStop();
		uiResettingStep := 300;
	300:
		IF ConveyorMotorA.InStopped AND 
			ConveyorMotorB.InStopped THEN
		//	DAS.fbStorageArea.M_InactivePulloutConveyorInternCtrl();
			uiResettingStep := 9000;
		END_IF
	9000:
		_Error :=false;
		 Error :=false;
		_ResetCompleted := TRUE;
END_CASE
IF _ResetCompleted THEN
	eState := STATE_DORMANT;
END_IF
END_METHOD

END_FUNCTION_BLOCK

// ---- Library/20_MachineUnits/22_AllocateArea/Old_Version_Service/FB_PullOutConveyorBtnCtrl_OLD.TcPOU
FUNCTION_BLOCK FB_PullOutConveyorBtnCtrl_OLD 
VAR_INPUT
	Input	:REFERENCE TO ST_InputTable;
	Output	:REFERENCE TO ST_OutputTable;
//	ConveyorMotorA :REFERENCE TO FB_Motor;
//	ConveyorMotorB :REFERENCE TO FB_Motor;
	Motor	:REFERENCE TO UNI_MotorList;
	
	
	bPullOutConveyorExecute	:BOOL;
	bPullOutConveyorDone	:BOOL;
	bPullOutConveyorBusy	:BOOL;
	StroageRegionMode :E_UnitMode ;
END_VAR
VAR_OUTPUT
	PullOutConveyorState :E_PullOutConveyorState;
END_VAR
VAR
	ExecutingStep	:E_PullOutConveyorState;
	bReferenceComponetIsRefed :BOOL;
	Forward_EdgeDetect	:FB_EdgeDetect;
	Backward_EdgeDetect	:FB_EdgeDetect;
END_VAR

clcUpdate();
Forward_EdgeDetect(xInput:=Input.bPullOutCV_FwdPb);
Backward_EdgeDetect(xInput :=Input.bPullOutCV_RevPb);
//IF __ISVALIDREF(BtnMoveForward) AND
//	__ISVALIDREF(BtnMoveReverse) AND
//	__ISVALIDREF(ConveyorMotorA) AND
//	__ISVALIDREF(ConveyorMotorB) THEN
	
//	bReferenceComponetIsRefed :=TRUE;
//END_IF

//IF bReferenceComponetIsRefed THEN
//	clcUpdate();
//END_IF

METHOD PRIVATE clcUpdate : BOOL
VAR_INPUT
END_VAR

CASE ExecutingStep OF
	E_PullOutConveyorState.idle:
	;
	
	E_PullOutConveyorState.AutoMode:
		M_TurnOff();
		M_TurnOff();
			IF bPullOutConveyorDone AND 
				NOT bPullOutConveyorExecute AND 
				NOT (StroageRegionMode = E_MachineMode.AUTO)  THEN
				ExecutingStep := E_PullOutConveyorState.Free;
			END_IF
	
	E_PullOutConveyorState.Free:
		M_TurnOn();
		M_TurnOn();
		IF NOT (StroageRegionMode = E_UnitMode.AUTO) AND 
				(StroageRegionMode = E_UnitMode.MANUAL) THEN
//			IF BtnMoveReverse.P_ButtonState AND BtnMoveForward.P_ButtonState THEN
			IF Input.bPullOutCV_FwdPb AND Input.bPullOutCV_RevPb THEN
//				ConveyorMotorA.M_StopMotor('');
//				ConveyorMotorB.M_StopMotor('');
				Motor.List.PullOutCV_A.M_MotorStop();
				Motor.List.PullOutCV_B.M_MotorStop();
					ELSIF Forward_EdgeDetect.xFallingEdge THEN 
						Motor.List.PullOutCV_A.M_MotorStop();
						Motor.List.PullOutCV_B.M_MotorStop();
					ELSIF Backward_EdgeDetect.xFallingEdge THEN
						Motor.List.PullOutCV_A.M_MotorStop();
						Motor.List.PullOutCV_B.M_MotorStop();
					ELSIF Input.bPullOutCV_RevPb THEN
							Motor.List.PullOutCV_A.M_MoveBackward();
							Motor.List.PullOutCV_B.M_MoveBackward();
					ELSIF Input.bPullOutCV_FwdPb  THEN
							Motor.List.PullOutCV_A.M_MoveForward();
							Motor.List.PullOutCV_B.M_MoveForward();					
			END_IF
		END_IF
END_CASE

IF (bPullOutConveyorExecute AND bPullOutConveyorBusy ) OR (StroageRegionMode = E_UnitMode.AUTO)  THEN
	ExecutingStep := E_PullOutConveyorState.AutoMode;
ELSE
	ExecutingStep := E_PullOutConveyorState.Free;
END_IF

PullOutConveyorState:=ExecutingStep;
END_METHOD

METHOD PRIVATE M_TurnOff : BOOL
VAR_INPUT
END_VAR
Output.bPullOutCV_FwdPbLamp:=FALSE;
Output.bPullOutCV_RevPbLamp:=FALSE;
END_METHOD

METHOD PRIVATE M_TurnOn : BOOL
VAR_INPUT
END_VAR
Output.bPullOutCV_FwdPbLamp:=TRUE;
Output.bPullOutCV_RevPbLamp:=TRUE;
END_METHOD

END_FUNCTION_BLOCK
